FUNCTION F_ToAnyInt : T_AnyInt
VAR_INPUT
    anyInt	: ANY_INT;
END_VAR

F_ToAnyInt := anyInt;

END_FUNCTION

(* stored: Version 1.1.0.1
   POU F_ToAnyInt: Id {85274dfa-47f8-4797-aeaa-1a54bdacdf07}, SpecialFunc None *)
